Fanuc KAREL source: kt00178.KL

-- PROVISIONAL review KL for V770-1; original PC SHA256 02393a03f3d06c3ebb3b44be1395b8ce36a0d39aeac7f69d7fd865a41cef202c
-- Incomplete behavior may be omitted. Consult companion uncertainty JSON. Do not deploy.
PROGRAM KT00178
%NOLOCKGROUP
VAR
  I2 : INTEGER
  OUT : REAL
-- UNRESOLVED_DECL Y1 type=002018
BEGIN
  -- UNRESOLVED_PC offsets 5-19; opcodes 2E,22,9D,33,B2
  -- UNRESOLVED_PC offsets 24-35; opcodes 2E,23
  -- UNRESOLVED_PC offsets 40-63; opcodes 22,9D,33,B1,21,56,64,23
  -- UNRESOLVED_PC offsets 68-72; opcodes 7F
END KT00178
